# B&R Automation Studio project LoteadorPractica
Automation Studio 4.12.5.95 SP; technology packages: mapp 5.24.3

## Configuration Config1

CPU 4PPC30.0702-23B, AutomationRuntime M4.93, Build 4.1.2, Vc V4.73.3

### Task classes (Cpu.sw)
```
Cyclic#1 (cycle 10000 us, tolerance 10000 us):
  LoteCtrl <- Source.Control.LoteCtrl.prg
Cyclic#4 (cycle 100000 us, tolerance 100000 us):
  VisuCtrl <- Source.Visu.VisuCtrl.prg
VcDataObjects: Visu1 <- Source.Visu.Visu1.dob
Binaries: vccdt, vccbmp, vccline, vcfile, arial, vctcal, vcrt, vcmgr, arsvcreg, vccstr, vcbclass, vccbtn, vcgclass, vcnet, vccscale, vcchtml, vcdsint, arflatprv, vcshared, vcclbox, vccddbox, arialbd, vcxml, vccnum, vcpdvnc, FWRules, arcoal, vccalarm, vccurl, vccslider, Visu101, vcchspot, vccpiech, Visu103, vcpdsw, vcfntttf, vccovl, vccshape, vcalarm, vcpkat, vcctext, vcctrend, udbdef, vccpopup, vcpfar00, vcdsloc, Visu102, TCData, arconfig, UserLog, AlarmSys, RecipeCore, AlarmHist, asfw, FileExplo, iomap, Role, ashwd, ashwac, sysconf, Users, User
Libraries: MpAlarmX, MpBase, astime, runtime, MpFile, FileIO, MpRecipe, sys_lib, MpUserX, MpCom, asieccon, asbrstr, asusb, aseth, ashw, dataobj, arcert, aruser, vcresman
```

### Hardware
```
4PPC30_0702_23B : 4PPC30.0702-23B v1.1.3.0
  Connector IF3:
    ActivateDevice = 1
    Mode = Manual
    InternetAddress = 192.168.150.95
    SubnetMask = 255.255.255.0
    Vnc1
    VncVcObjectName1 = Visu1
    VncKeyMappingFile1 = VC\PS2-Keyboard.dis
    ActivateSnmp = 2
  ConfigurationID = LoteadorPractica_Config1
  TimerDeviceType = SWIOTIMER
  Cyclic1Duration = 10000
  Cyclic1Tolerance = 10000
  Cyclic2Duration = 20000
  Cyclic2Tolerance = 20000
  Cyclic3Duration = 50000
  Cyclic3Tolerance = 50000
  Cyclic4Duration = 100000
  Cyclic4Tolerance = 100000
  Cyclic5Duration = 200000
  Cyclic5Tolerance = 200000
  Cyclic6Duration = 500000
  Cyclic6Tolerance = 500000
  Cyclic7Duration = 1000000
  Cyclic7Tolerance = 1000000
  Cyclic8Duration = 10000
  Cyclic8Tolerance = 30000000
  FileDevice1
  FileDeviceName1 = USER
  FileDevicePath1 = USER_PATH
  KeyMappingFile = VC\4PPC30_0702_23B.dis
```

## Logical view

Binary libraries used (declarations not repeated): operator, runtime, astime, AsIecCon, MpAlarmX, MpBase, MpFile, FileIO, MpRecipe, sys_lib, MpUserX, MpCom

### Global.typ - Global data types
```iecst
(**********************************  ESTRUCTURA DE MAQUINA GLOBAL *********************************)
(***********************************************************************************************************************)

TYPE
	Machine_ctrl_type : 	STRUCT
		cmd : Machine_cmd_type;
		param : Machine_param_type;
		status : Machine_status_type;
		state : Machine_state_type;
	END_STRUCT;
	Machine_cmd_type : 	STRUCT
	END_STRUCT;
	Machine_param_type : 	STRUCT
	END_STRUCT;
	Machine_status_type : 	STRUCT
	END_STRUCT;
	Machine_state_type : 	STRUCT
	END_STRUCT;
END_TYPE

(**********************************  ESTRUCTURA DE VARIABLES REMANENTES *********************************)
(***********************************************************************************************************************)

TYPE
	Machine_remanent_type : 	STRUCT
	END_STRUCT;
END_TYPE

(**********************************  ESTRUCTURA DE VISU *********************************)
(***********************************************************************************************************************)

TYPE
	Visu_type : 	STRUCT
		buttons : Visu_buttons_type;
		numInputs : Visu_numInputs_type;
		numOutputs : Visu_numOutputs_type;
	END_STRUCT;
	Visu_buttons_type : 	STRUCT
		buttonAddToList : BOOL;
	END_STRUCT;
	Visu_numInputs_type : 	STRUCT
		batch : UINT;
		material : STRING[80];
	END_STRUCT;
	Visu_numOutputs_type : 	STRUCT
		New_Member : USINT;
	END_STRUCT;
END_TYPE
```

### Global.var - Global variables
```iecst
VAR
	gCtrl : Machine_ctrl_type;
	gVisu : Visu_type;
END_VAR
VAR RETAIN
	gRemanentParam : {REDUND_UNREPLICABLE} Machine_remanent_type;
END_VAR
```

### Constants.var
```iecst
(***********************************CONSTANTES DE NUMERO DE LOTES********************************************************************)
VAR CONSTANT
	MAX_NUM_BATCH : USINT := 10;
END_VAR
```


### Program Logical/Source/Control/LoteCtrl (IEC)

#### Main.st - Init, cyclic, exit code
```iecst
PROGRAM _INIT
	(* Insert code here *)

END_PROGRAM

PROGRAM _CYCLIC
	//VARIABLES GLOBALES A LOCALES

	//*****************************CONDICIONES************************************************************
	FOR i := 1 TO MAX_NUM_BATCH DO
		IF LoteCtrl.param.numberBatch[i] > 0 THEN
			LoteCtrl.status.writtenLine[i] := TRUE;
		ELSE
			LoteCtrl.status.writtenLine[i] := FALSE;
		END_IF;
//		LoteCtrl.status.numberBatch[i] := gVisu.numInputs.batch;

	 	IF  EDGEPOS(gVisu.buttons.buttonAddToList) THEN
//		FOR i := 1 TO MAX_NUM_BATCH DO
//			LoteCtrl.status.numberBatch[i] := gVisu.numInputs.batch;
//
//		END_FOR;
			IF NOT (LoteCtrl.status.writtenLine[1])  THEN
				LoteCtrl.param.numberBatch[1] := gVisu.numInputs.batch;

			END_IF;

			IF  (LoteCtrl.status.writtenLine[1]) AND NOT (LoteCtrl.status.writtenLine[2])  THEN
				LoteCtrl.param.numberBatch[2] := gVisu.numInputs.batch;

			END_IF;

			IF  (LoteCtrl.status.writtenLine[2]) AND NOT (LoteCtrl.status.writtenLine[3]) THEN
				LoteCtrl.param.numberBatch[3] := gVisu.numInputs.batch;

			END_IF;

			IF  (LoteCtrl.status.writtenLine[3]) AND NOT (LoteCtrl.status.writtenLine[4]) THEN
				LoteCtrl.param.numberBatch[4] := gVisu.numInputs.batch;

			END_IF;

			IF  (LoteCtrl.status.writtenLine[4]) AND NOT (LoteCtrl.status.writtenLine[5]) THEN
				LoteCtrl.param.numberBatch[5] := gVisu.numInputs.batch;

			END_IF;

			IF  (LoteCtrl.status.writtenLine[5]) AND NOT (LoteCtrl.status.writtenLine[6]) THEN
				LoteCtrl.param.numberBatch[6] := gVisu.numInputs.batch;

			END_IF;

			IF  (LoteCtrl.status.writtenLine[6]) AND NOT (LoteCtrl.status.writtenLine[7]) THEN
				LoteCtrl.param.numberBatch[7] := gVisu.numInputs.batch;

			END_IF;

			IF  (LoteCtrl.status.writtenLine[7]) AND NOT (LoteCtrl.status.writtenLine[8]) THEN
				LoteCtrl.param.numberBatch[8] := gVisu.numInputs.batch;

			END_IF;

			IF  (LoteCtrl.status.writtenLine[8]) AND NOT (LoteCtrl.status.writtenLine[9]) THEN
				LoteCtrl.param.numberBatch[9] := gVisu.numInputs.batch;

			END_IF;

			IF  (LoteCtrl.status.writtenLine[9]) AND NOT (LoteCtrl.status.writtenLine[10]) THEN
				LoteCtrl.param.numberBatch[10] := gVisu.numInputs.batch;

			END_IF;

		END_IF;

	END_FOR;
END_PROGRAM

PROGRAM _EXIT
	(* Insert code here *)

END_PROGRAM
```

#### Types.typ - Local data types
```iecst
TYPE
	LoteCtrl_type : 	STRUCT
		cmd : LoteCtrl_cmd_type;
		param : LoteCtrl_param_type;
		status : LoteCtrl_status_type;
		state : LoteCtrl_state_type;
	END_STRUCT;
	LoteCtrl_cmd_type : 	STRUCT
		New_Member : USINT;
	END_STRUCT;
	LoteCtrl_param_type : 	STRUCT
		numberBatch : ARRAY[1..MAX_NUM_BATCH]OF UINT;
	END_STRUCT;
	LoteCtrl_status_type : 	STRUCT
		writtenLine : ARRAY[1..MAX_NUM_BATCH]OF BOOL;
	END_STRUCT;
	LoteCtrl_state_type : 	STRUCT
		New_Member : USINT;
	END_STRUCT;
END_TYPE
```

#### Variables.var - Local variables
```iecst
VAR
	LoteCtrl : LoteCtrl_type;
	i : USINT;
END_VAR
```

#### ActionTime.st
```iecst
ACTION ActionTime:

(*Lee la hora y la fecha del reloj de tiempo real y escribe esta información en una estructura RTCtime_struct.*)

	status_gettime := RTC_gettime(ADR(rtc_gettime)); (* get current time and store it into time struct *)

	//	status_settime := RTC_settime(ADR(rtc_settime));

	//	IF ((rtc_gettime.hour = 12) AND (rtc_gettime.minute >= 0) AND (rtc_gettime.minute <= 30)) THEN (* check time interval *)
	//		DOUT1 := 1; (* set output to high *)
	//	ELSE
	//		DOUT1 := 0; (* set output to low *)
	//	END_IF

(*Lee la hora y la fecha del reloj de tiempo real y escribe esta información en una estructura RTCtime_struct. *)

	rtc_settime.year 		:= 2025;
	rtc_settime.month 		:= rtc_gettime.month;
	rtc_settime.day 		:= rtc_gettime.day;
	rtc_settime.hour 		:= rtc_gettime.hour;
	rtc_settime.minute 		:= rtc_gettime.minute;
	rtc_settime.second 		:= rtc_gettime.second;
	rtc_settime.millisec 	:= rtc_gettime.millisec;

	//	rtc_gettime.millisec := rtc_gettime.millisec +1;
	//	IF rtc_gettime.millisec >= 100 THEN
	//		rtc_gettime.millisec := 0;
	//	  rtc_gettime.second := rtc_gettime.second +1;
	//	END_IF;
	//
	//	IF rtc_gettime.second >= 60 THEN
	//		rtc_gettime.second := 0;
	//		rtc_gettime.minute := rtc_gettime.minute +1;
	//	END_IF;
	//
	//	IF rtc_gettime.minute >= 60 THEN
	//		rtc_gettime.minute := 0;
	//		rtc_gettime.hour := rtc_gettime.hour +1;
	//	END_IF;
	//
	//	IF rtc_gettime.hour >= 24 THEN
	//		rtc_gettime.hour := 0;
	//		rtc_gettime.day := rtc_gettime.day +1;
	//	END_IF;

END_ACTION
```

- Visualisation Logical/Source/Visu (not shown)
